// TIA Portal V19 export
DATA_BLOCK "DB Mauvaises Pièces"   // DB13
// stored: AutoNumber false
   VAR RETAIN
      "Nb_J-1" : Int;
      "Nb_J-2" : Int;
      "Nb_J-3" : Int;
      "Nb_J-4" : Int;
      "Nb_J-5" : Int;
      "Nb_J-6" : Int;
      "Nb_J-7" : Int;
      "Nb_J-8" : Int;
      "Nb_J-9" : Int;
      "Nb_J-10" : Int;
      "Nb_J-11" : Int;
      "Nb_J-12" : Int;
      "Nb_J-13" : Int;
      "Nb_J-14" : Int;
      "Nb_J-15" : Int;
      "Nb_J-16" : Int;
      "Nb_J-17" : Int;
      "Nb_J-18" : Int;
      "Nb_J-19" : Int;
      "Nb_J-20" : Int;
      "Nb_J-21" : Int;
      "Nb_J-22" : Int;
      "Nb_J-23" : Int;
      "Nb_J-24" : Int;
      "Nb_J-25" : Int;
      "Nb_J-26" : Int;
      "Nb_J-27" : Int;
      "Nb_J-28" : Int;
      "Nb_J-29" : Int;
      "Nb_J-30" : Int;
      "Nb_J-31" : Int;
   END_VAR
BEGIN
END_DATA_BLOCK
